(*

.. <legal notes>

legal notes
=================
| SPDX-FileCopyrightText: © 2026 Oleksandr Tiutyk <trofimich@gmail.com>
| SPDX-License-Identifier: LGPL-3.0-only
| For details check: LGPL-3.0-only_

.. _LGPL-3.0-only: https://www.gnu.org/licenses/lgpl-3.0.en.html

.. </legal notes>

*)

INTERFACE IAutomationControllerPlugin EXTENDS __SYSTEM.IQueryInterface

METHOD OnAfterControllerExecute
VAR_INPUT
	controller : IAutomationController;
END_VAR
END_METHOD

METHOD OnBeforeControllerExecute
VAR_INPUT
	controller : IAutomationController;
END_VAR
END_METHOD

END_INTERFACE

(* stored: Version 1.1.0.1
   Itf IAutomationControllerPlugin: Id {11f4ca86-c242-4443-b1d6-97f70e22041e}
   Method OnAfterControllerExecute: Id {74692b1f-e693-4fbd-b9c0-cccf39583549}
   Method OnBeforeControllerExecute: Id {e34f4211-71a0-47a6-9215-681c63206f5c} *)
